		//Wait for Delay, copy Data and then next step
		IF NOT fbMBRead_FC3.bBusy AND NOT fbMBRead_FC3.bError AND timDelay.Q THEN
			// convert received data
			FB_ConvertData(	arrBuffer_FC3			:=	arrBuffer_FC3,
											int_Poll_Counter		:=	int_Poll_Counter,
											lrPowerTotal			=>	fbMeter[int_Poll_Counter].lrPowerTotal,	
											lrReactivePowerTotal	=> 	fbMeter[int_Poll_Counter].lrReactivePowerTotal,
											eOperatingStateInverter	=>	st_Huawei_SmartLogger[int_Poll_Counter].eOperatingStateInverter);
	
			//Next Step
			fbMBRead_FC3.bExecute := FALSE;
			timDelay.IN := FALSE;
			iStateModbus := iStateModbus+1;
			IF arrBuffer_FC3[9]<>0 THEN
				st_Huawei_SmartLogger[int_Poll_Counter].bError := FALSE; 
				st_Huawei_SmartLogger[int_Poll_Counter].eErrorState := E_Huawei_SmartLogger_Error.eNoError;
			ELSE
				st_Huawei_SmartLogger[int_Poll_Counter].bError := FALSE; 
				st_Huawei_SmartLogger[int_Poll_Counter].eErrorState := E_Huawei_SmartLogger_Error.eNoError;
			END_IF
		END_IF
			
		//Error from Inverter 
		IF NOT fbMBRead_FC3.bBusy AND NOT fbMBRead_FC3.bError AND timDelay.Q AND arrBuffer_FC3[9] >= 16#0300 AND arrBuffer_FC3[9] <= 16#0308 THEN
			iStateModbus := 300;
			st_Huawei_SmartLogger[int_Poll_Counter].eErrorState := E_Huawei_SmartLogger_Error.eHuawei_SmartLoggerError;
		END_IF
	
		//Error or Timeout
		IF FPError_FC_3.Q OR timTimeout.Q THEN
			iStateModbus := 300;
			st_Huawei_SmartLogger[int_Poll_Counter].eOperatingStateInverter := E_Huawei_SmartLogger_OperatingState.Unknown;
			st_Huawei_SmartLogger[int_Poll_Counter].eErrorState	:=	E_Huawei_SmartLogger_Error.eModbusTCPError;
		END_IF
		
	2://Wait and go to step 1 or step 3
		iStateModbus_CP := iStateModbus;
		IF sint_ID_Iverter[int_Poll_Counter+1] = 0 OR int_Poll_Counter=int_maxPolls THEN		// if ID is not in use, go to state 100
			iStateModbus := 100;
		ELSE
			iStateModbus := 3;
			int_Poll_Counter:=int_Poll_Counter+1;			//Poll int_Poll_Counter : Inverter int_Poll_Counter 	
		END_IF

	3://Read out next inverter
		st_Huawei_SmartLogger[int_Poll_Counter].bFunctionIsActive := TRUE;
		iStateModbus_CP := iStateModbus;
		fbMBRead_FC3.nQuantity := 25;
		fbMBRead_FC3.nMBAddr := (51000+(25*(SINT_TO_WORD(sint_ID_Iverter[int_Poll_Counter]) - 1)));
		fbMBRead_FC3.bExecute := TRUE;
			
		IF fbMBRead_FC3.bBusy THEN 
			timDelay.IN := TRUE; 
		END_IF
		
		//Wait for Delay, copy Data and then next step
		IF NOT fbMBRead_FC3.bBusy AND NOT fbMBRead_FC3.bError AND timDelay.Q THEN
			// convert received data
			FB_ConvertData(	arrBuffer_FC3			:=	arrBuffer_FC3,
											int_Poll_Counter		:=	int_Poll_Counter,
											lrPowerTotal			=>	fbMeter[int_Poll_Counter].lrPowerTotal,	
											lrReactivePowerTotal	=> 	fbMeter[int_Poll_Counter].lrReactivePowerTotal,
											eOperatingStateInverter	=>	st_Huawei_SmartLogger[int_Poll_Counter].eOperatingStateInverter);
	
			//Next Step
			fbMBRead_FC3.bExecute := FALSE;
			timDelay.IN := FALSE;
			iStateModbus := iStateModbus+1;
			IF arrBuffer_FC3[9]<>0 THEN
				st_Huawei_SmartLogger[int_Poll_Counter].bError := FALSE; 
				st_Huawei_SmartLogger[int_Poll_Counter].eErrorState := E_Huawei_SmartLogger_Error.eNoError;
			ELSE
				st_Huawei_SmartLogger[int_Poll_Counter].bError := FALSE; 
				st_Huawei_SmartLogger[int_Poll_Counter].eErrorState := E_Huawei_SmartLogger_Error.eNoError;
			END_IF
		END_IF
			
		//Error from Inverter 
		IF NOT fbMBRead_FC3.bBusy AND NOT fbMBRead_FC3.bError AND timDelay.Q AND arrBuffer_FC3[9] >= 16#0300 AND arrBuffer_FC3[9] <= 16#0308 THEN
			iStateModbus := 300;
			st_Huawei_SmartLogger[int_Poll_Counter].eErrorState := E_Huawei_SmartLogger_Error.eHuawei_SmartLoggerError;
		END_IF
	
		//Error or Timeout
		IF FPError_FC_3.Q OR timTimeout.Q THEN
			iStateModbus := 300;
			st_Huawei_SmartLogger[int_Poll_Counter].eOperatingStateInverter := E_Huawei_SmartLogger_OperatingState.Unknown;
			st_Huawei_SmartLogger[int_Poll_Counter].eErrorState	:=	E_Huawei_SmartLogger_Error.eModbusTCPError;
		END_IF
		
	4://Wait and go to step +1 or step 100
		iStateModbus_CP := iStateModbus;
		IF sint_ID_Iverter[int_Poll_Counter+1] = 0 OR int_Poll_Counter=int_maxPolls THEN		// if ID is not in use, go to state 100
			iStateModbus := 100;
		ELSE
			iStateModbus := iStateModbus+1;
			int_Poll_Counter:=int_Poll_Counter+1;			//Poll int_Poll_Counter : Inverter int_Poll_Counter 	
		END_IF
	
	5://Read out next inverter
		st_Huawei_SmartLogger[int_Poll_Counter].bFunctionIsActive := TRUE;
		iStateModbus_CP := iStateModbus;
		fbMBRead_FC3.nQuantity := 25;
		fbMBRead_FC3.nMBAddr := (51000+(25*(SINT_TO_WORD(sint_ID_Iverter[int_Poll_Counter]) - 1)));
		fbMBRead_FC3.bExecute := TRUE;
			
		IF fbMBRead_FC3.bBusy THEN 
			timDelay.IN := TRUE; 
		END_IF
		
		//Wait for Delay, copy Data and then next step
		IF NOT fbMBRead_FC3.bBusy AND NOT fbMBRead_FC3.bError AND timDelay.Q THEN
			// convert received data
			FB_ConvertData(	arrBuffer_FC3			:=	arrBuffer_FC3,
											int_Poll_Counter		:=	int_Poll_Counter,
											lrPowerTotal			=>	fbMeter[int_Poll_Counter].lrPowerTotal,	
											lrReactivePowerTotal	=> 	fbMeter[int_Poll_Counter].lrReactivePowerTotal,
											eOperatingStateInverter	=>	st_Huawei_SmartLogger[int_Poll_Counter].eOperatingStateInverter);
	
			//Next Step
			fbMBRead_FC3.bExecute := FALSE;
			timDelay.IN := FALSE;
			iStateModbus := iStateModbus+1;
			IF arrBuffer_FC3[9]<>0 THEN
				st_Huawei_SmartLogger[int_Poll_Counter].bError := FALSE; 
				st_Huawei_SmartLogger[int_Poll_Counter].eErrorState := E_Huawei_SmartLogger_Error.eNoError;
			ELSE
				st_Huawei_SmartLogger[int_Poll_Counter].bError := FALSE; 
				st_Huawei_SmartLogger[int_Poll_Counter].eErrorState := E_Huawei_SmartLogger_Error.eNoError;
			END_IF
		END_IF
			
		//Error from Inverter 
		IF NOT fbMBRead_FC3.bBusy AND NOT fbMBRead_FC3.bError AND timDelay.Q AND arrBuffer_FC3[9] >= 16#0300 AND arrBuffer_FC3[9] <= 16#0308 THEN
			iStateModbus := 300;
			st_Huawei_SmartLogger[int_Poll_Counter].eErrorState := E_Huawei_SmartLogger_Error.eHuawei_SmartLoggerError;
		END_IF
	
		//Error or Timeout
		IF FPError_FC_3.Q OR timTimeout.Q THEN
			iStateModbus := 300;
			st_Huawei_SmartLogger[int_Poll_Counter].eOperatingStateInverter := E_Huawei_SmartLogger_OperatingState.Unknown;
			st_Huawei_SmartLogger[int_Poll_Counter].eErrorState	:=	E_Huawei_SmartLogger_Error.eModbusTCPError;
		END_IF
		
	6://Wait and go to step +1 or step 100
		iStateModbus_CP := iStateModbus;
		IF sint_ID_Iverter[int_Poll_Counter+1] = 0 OR int_Poll_Counter=int_maxPolls THEN		// if ID is not in use, go to state 100
			iStateModbus := 100;
		ELSE
			iStateModbus := iStateModbus+1;
			int_Poll_Counter:=int_Poll_Counter+1;			//Poll int_Poll_Counter : Inverter int_Poll_Counter 	
		END_IF
		
	7://Read out next inverter
		st_Huawei_SmartLogger[int_Poll_Counter].bFunctionIsActive := TRUE;
		iStateModbus_CP := iStateModbus;
		fbMBRead_FC3.nQuantity := 25;
		fbMBRead_FC3.nMBAddr := (51000+(25*(SINT_TO_WORD(sint_ID_Iverter[int_Poll_Counter]) - 1)));
		fbMBRead_FC3.bExecute := TRUE;
			
		IF fbMBRead_FC3.bBusy THEN 
			timDelay.IN := TRUE; 
		END_IF
		
		//Wait for Delay, copy Data and then next step
		IF NOT fbMBRead_FC3.bBusy AND NOT fbMBRead_FC3.bError AND timDelay.Q THEN
			// convert received data
			FB_ConvertData(	arrBuffer_FC3			:=	arrBuffer_FC3,
											int_Poll_Counter		:=	int_Poll_Counter,
											lrPowerTotal			=>	fbMeter[int_Poll_Counter].lrPowerTotal,	
											lrReactivePowerTotal	=> 	fbMeter[int_Poll_Counter].lrReactivePowerTotal,
											eOperatingStateInverter	=>	st_Huawei_SmartLogger[int_Poll_Counter].eOperatingStateInverter);
	
			//Next Step
			fbMBRead_FC3.bExecute := FALSE;
			timDelay.IN := FALSE;
			iStateModbus := iStateModbus+1;
			IF arrBuffer_FC3[9]<>0 THEN
				st_Huawei_SmartLogger[int_Poll_Counter].bError := FALSE; 
				st_Huawei_SmartLogger[int_Poll_Counter].eErrorState := E_Huawei_SmartLogger_Error.eNoError;
			ELSE
				st_Huawei_SmartLogger[int_Poll_Counter].bError := FALSE; 
				st_Huawei_SmartLogger[int_Poll_Counter].eErrorState := E_Huawei_SmartLogger_Error.eNoError;
			END_IF
		END_IF
			
		//Error from Inverter 
		IF NOT fbMBRead_FC3.bBusy AND NOT fbMBRead_FC3.bError AND timDelay.Q AND arrBuffer_FC3[9] >= 16#0300 AND arrBuffer_FC3[9] <= 16#0308 THEN
			iStateModbus := 300;
			st_Huawei_SmartLogger[int_Poll_Counter].eErrorState := E_Huawei_SmartLogger_Error.eHuawei_SmartLoggerError;
		END_IF
	
		//Error or Timeout
		IF FPError_FC_3.Q OR timTimeout.Q THEN
			iStateModbus := 300;
			st_Huawei_SmartLogger[int_Poll_Counter].eOperatingStateInverter := E_Huawei_SmartLogger_OperatingState.Unknown;
			st_Huawei_SmartLogger[int_Poll_Counter].eErrorState	:=	E_Huawei_SmartLogger_Error.eModbusTCPError;
		END_IF

	8://Wait and go to step +1 or step 100
		iStateModbus_CP := iStateModbus;
		IF sint_ID_Iverter[int_Poll_Counter+1] = 0 OR int_Poll_Counter=int_maxPolls THEN		// if ID is not in use, go to state 100
			iStateModbus := 100;
		ELSE
			iStateModbus := iStateModbus+1;
			int_Poll_Counter:=int_Poll_Counter+1;			//Poll int_Poll_Counter : Inverter int_Poll_Counter 	
		END_IF
		
	9://Read out next inverter
		st_Huawei_SmartLogger[int_Poll_Counter].bFunctionIsActive := TRUE;
		iStateModbus_CP := iStateModbus;
		fbMBRead_FC3.nQuantity := 25;
		fbMBRead_FC3.nMBAddr := (51000+(25*(SINT_TO_WORD(sint_ID_Iverter[int_Poll_Counter]) - 1)));
		fbMBRead_FC3.bExecute := TRUE;
			
		IF fbMBRead_FC3.bBusy THEN 
			timDelay.IN := TRUE; 
		END_IF
		
		//Wait for Delay, copy Data and then next step
		IF NOT fbMBRead_FC3.bBusy AND NOT fbMBRead_FC3.bError AND timDelay.Q THEN
			// convert received data
			FB_ConvertData(	arrBuffer_FC3			:=	arrBuffer_FC3,
											int_Poll_Counter		:=	int_Poll_Counter,
											lrPowerTotal			=>	fbMeter[int_Poll_Counter].lrPowerTotal,	
											lrReactivePowerTotal	=> 	fbMeter[int_Poll_Counter].lrReactivePowerTotal,
											eOperatingStateInverter	=>	st_Huawei_SmartLogger[int_Poll_Counter].eOperatingStateInverter);
	
			//Next Step
			fbMBRead_FC3.bExecute := FALSE;
			timDelay.IN := FALSE;
			iStateModbus := iStateModbus+1;
			IF arrBuffer_FC3[9]<>0 THEN
				st_Huawei_SmartLogger[int_Poll_Counter].bError := FALSE; 
				st_Huawei_SmartLogger[int_Poll_Counter].eErrorState := E_Huawei_SmartLogger_Error.eNoError;
			ELSE
				st_Huawei_SmartLogger[int_Poll_Counter].bError := FALSE; 
				st_Huawei_SmartLogger[int_Poll_Counter].eErrorState := E_Huawei_SmartLogger_Error.eNoError;
			END_IF
		END_IF
			
		//Error from Inverter 
		IF NOT fbMBRead_FC3.bBusy AND NOT fbMBRead_FC3.bError AND timDelay.Q AND arrBuffer_FC3[9] >= 16#0300 AND arrBuffer_FC3[9] <= 16#0308 THEN
			iStateModbus := 300;
			st_Huawei_SmartLogger[int_Poll_Counter].eErrorState := E_Huawei_SmartLogger_Error.eHuawei_SmartLoggerError;
		END_IF
	
		//Error or Timeout
		IF FPError_FC_3.Q OR timTimeout.Q THEN
			iStateModbus := 300;
			st_Huawei_SmartLogger[int_Poll_Counter].eOperatingStateInverter := E_Huawei_SmartLogger_OperatingState.Unknown;
			st_Huawei_SmartLogger[int_Poll_Counter].eErrorState	:=	E_Huawei_SmartLogger_Error.eModbusTCPError;
		END_IF
		
	10://Wait and go to step +1 or step 100
		iStateModbus_CP := iStateModbus;
		IF sint_ID_Iverter[int_Poll_Counter+1] = 0 OR int_Poll_Counter=int_maxPolls THEN		// if ID is not in use, go to state 100
			iStateModbus := 100;
		ELSE
			iStateModbus := iStateModbus+1;
			int_Poll_Counter:=int_Poll_Counter+1;			//Poll int_Poll_Counter : Inverter int_Poll_Counter 	
		END_IF
		
	11://Read out next inverter
		st_Huawei_SmartLogger[int_Poll_Counter].bFunctionIsActive := TRUE;
		iStateModbus_CP := iStateModbus;
		fbMBRead_FC3.nQuantity := 25;
		fbMBRead_FC3.nMBAddr := (51000+(25*(SINT_TO_WORD(sint_ID_Iverter[int_Poll_Counter]) - 1)));
		fbMBRead_FC3.bExecute := TRUE;
			
		IF fbMBRead_FC3.bBusy THEN 
			timDelay.IN := TRUE; 
		END_IF
		
		//Wait for Delay, copy Data and then next step
		IF NOT fbMBRead_FC3.bBusy AND NOT fbMBRead_FC3.bError AND timDelay.Q THEN
			// convert received data
			FB_ConvertData(	arrBuffer_FC3			:=	arrBuffer_FC3,
											int_Poll_Counter		:=	int_Poll_Counter,
											lrPowerTotal			=>	fbMeter[int_Poll_Counter].lrPowerTotal,	
											lrReactivePowerTotal	=> 	fbMeter[int_Poll_Counter].lrReactivePowerTotal,
											eOperatingStateInverter	=>	st_Huawei_SmartLogger[int_Poll_Counter].eOperatingStateInverter);
	
			//Next Step
			fbMBRead_FC3.bExecute := FALSE;
			timDelay.IN := FALSE;
			iStateModbus := iStateModbus+1;
			IF arrBuffer_FC3[9]<>0 THEN
				st_Huawei_SmartLogger[int_Poll_Counter].bError := FALSE; 
				st_Huawei_SmartLogger[int_Poll_Counter].eErrorState := E_Huawei_SmartLogger_Error.eNoError;
			ELSE
				st_Huawei_SmartLogger[int_Poll_Counter].bError := FALSE; 
				st_Huawei_SmartLogger[int_Poll_Counter].eErrorState := E_Huawei_SmartLogger_Error.eNoError;
			END_IF
		END_IF
			
		//Error from Inverter 
		IF NOT fbMBRead_FC3.bBusy AND NOT fbMBRead_FC3.bError AND timDelay.Q AND arrBuffer_FC3[9] >= 16#0300 AND arrBuffer_FC3[9] <= 16#0308 THEN
			iStateModbus := 300;
			st_Huawei_SmartLogger[int_Poll_Counter].eErrorState := E_Huawei_SmartLogger_Error.eHuawei_SmartLoggerError;
		END_IF
	
		//Error or Timeout
		IF FPError_FC_3.Q OR timTimeout.Q THEN
			iStateModbus := 300;
			st_Huawei_SmartLogger[int_Poll_Counter].eOperatingStateInverter := E_Huawei_SmartLogger_OperatingState.Unknown;
			st_Huawei_SmartLogger[int_Poll_Counter].eErrorState	:=	E_Huawei_SmartLogger_Error.eModbusTCPError;
		END_IF
		
	12://Wait and go to step +1 or step 100
		iStateModbus_CP := iStateModbus;
		IF sint_ID_Iverter[int_Poll_Counter+1] = 0 OR int_Poll_Counter=int_maxPolls THEN		// if ID is not in use, go to state 100
			iStateModbus := 100;
		ELSE
			iStateModbus := iStateModbus+1;
			int_Poll_Counter:=int_Poll_Counter+1;			//Poll int_Poll_Counter : Inverter int_Poll_Counter 	
		END_IF
		
	13://Read out next inverter
		st_Huawei_SmartLogger[int_Poll_Counter].bFunctionIsActive := TRUE;
		iStateModbus_CP := iStateModbus;
		fbMBRead_FC3.nQuantity := 25;
		fbMBRead_FC3.nMBAddr := (51000+(25*(SINT_TO_WORD(sint_ID_Iverter[int_Poll_Counter]) - 1)));
		fbMBRead_FC3.bExecute := TRUE;
			
		IF fbMBRead_FC3.bBusy THEN 
			timDelay.IN := TRUE; 
		END_IF
		
		//Wait for Delay, copy Data and then next step
		IF NOT fbMBRead_FC3.bBusy AND NOT fbMBRead_FC3.bError AND timDelay.Q THEN
			// convert received data
			FB_ConvertData(	arrBuffer_FC3			:=	arrBuffer_FC3,
											int_Poll_Counter		:=	int_Poll_Counter,
											lrPowerTotal			=>	fbMeter[int_Poll_Counter].lrPowerTotal,	
											lrReactivePowerTotal	=> 	fbMeter[int_Poll_Counter].lrReactivePowerTotal,
											eOperatingStateInverter	=>	st_Huawei_SmartLogger[int_Poll_Counter].eOperatingStateInverter);
	
			//Next Step
			fbMBRead_FC3.bExecute := FALSE;
			timDelay.IN := FALSE;
			iStateModbus := iStateModbus+1;
			IF arrBuffer_FC3[9]<>0 THEN
				st_Huawei_SmartLogger[int_Poll_Counter].bError := FALSE; 
				st_Huawei_SmartLogger[int_Poll_Counter].eErrorState := E_Huawei_SmartLogger_Error.eNoError;
			ELSE
				st_Huawei_SmartLogger[int_Poll_Counter].bError := FALSE; 
				st_Huawei_SmartLogger[int_Poll_Counter].eErrorState := E_Huawei_SmartLogger_Error.eNoError;
			END_IF
		END_IF
			
		//Error from Inverter 1
		IF NOT fbMBRead_FC3.bBusy AND NOT fbMBRead_FC3.bError AND timDelay.Q AND arrBuffer_FC3[9] >= 16#0300 AND arrBuffer_FC3[9] <= 16#0308 THEN
			iStateModbus := 300;
			st_Huawei_SmartLogger[int_Poll_Counter].eErrorState := E_Huawei_SmartLogger_Error.eHuawei_SmartLoggerError;
		END_IF
	
		//Error or Timeout
		IF FPError_FC_3.Q OR timTimeout.Q THEN
			iStateModbus := 300;
			st_Huawei_SmartLogger[int_Poll_Counter].eOperatingStateInverter := E_Huawei_SmartLogger_OperatingState.Unknown;
			st_Huawei_SmartLogger[int_Poll_Counter].eErrorState	:=	E_Huawei_SmartLogger_Error.eModbusTCPError;
		END_IF
		
	14://Wait and go to step +1 or step 100
		iStateModbus_CP := iStateModbus;
		IF sint_ID_Iverter[int_Poll_Counter+1] = 0 OR int_Poll_Counter=int_maxPolls THEN		// if ID is not in use, go to state 100
			iStateModbus := 100;
		ELSE
			iStateModbus := iStateModbus+1;
			int_Poll_Counter:=int_Poll_Counter+1;			//Poll int_Poll_Counter : Inverter int_Poll_Counter 	
		END_IF
		
	15://Read out next inverter
		st_Huawei_SmartLogger[int_Poll_Counter].bFunctionIsActive := TRUE;
		iStateModbus_CP := iStateModbus;
		fbMBRead_FC3.nQuantity := 25;
		fbMBRead_FC3.nMBAddr := (51000+(25*(SINT_TO_WORD(sint_ID_Iverter[int_Poll_Counter]) - 1)));
		fbMBRead_FC3.bExecute := TRUE;
			
		IF fbMBRead_FC3.bBusy THEN 
			timDelay.IN := TRUE; 
		END_IF
		
		//Wait for Delay, copy Data and then next step
		IF NOT fbMBRead_FC3.bBusy AND NOT fbMBRead_FC3.bError AND timDelay.Q THEN
			// convert received data
			FB_ConvertData(	arrBuffer_FC3			:=	arrBuffer_FC3,
											int_Poll_Counter		:=	int_Poll_Counter,
											lrPowerTotal			=>	fbMeter[int_Poll_Counter].lrPowerTotal,	
											lrReactivePowerTotal	=> 	fbMeter[int_Poll_Counter].lrReactivePowerTotal,
											eOperatingStateInverter	=>	st_Huawei_SmartLogger[int_Poll_Counter].eOperatingStateInverter);
	
			//Next Step
			fbMBRead_FC3.bExecute := FALSE;
			timDelay.IN := FALSE;
			iStateModbus := iStateModbus+1;
			IF arrBuffer_FC3[9]<>0 THEN
				st_Huawei_SmartLogger[int_Poll_Counter].bError := FALSE; 
				st_Huawei_SmartLogger[int_Poll_Counter].eErrorState := E_Huawei_SmartLogger_Error.eNoError;
			ELSE
				st_Huawei_SmartLogger[int_Poll_Counter].bError := FALSE; 
				st_Huawei_SmartLogger[int_Poll_Counter].eErrorState := E_Huawei_SmartLogger_Error.eNoError;
			END_IF
		END_IF
			
		//Error from Inverter 
		IF NOT fbMBRead_FC3.bBusy AND NOT fbMBRead_FC3.bError AND timDelay.Q AND arrBuffer_FC3[9] >= 16#0300 AND arrBuffer_FC3[9] <= 16#0308 THEN
			iStateModbus := 300;
			st_Huawei_SmartLogger[int_Poll_Counter].eErrorState := E_Huawei_SmartLogger_Error.eHuawei_SmartLoggerError;
		END_IF
	
		//Error or Timeout
		IF FPError_FC_3.Q OR timTimeout.Q THEN
			iStateModbus := 300;
			st_Huawei_SmartLogger[int_Poll_Counter].eOperatingStateInverter := E_Huawei_SmartLogger_OperatingState.Unknown;
			st_Huawei_SmartLogger[int_Poll_Counter].eErrorState	:=	E_Huawei_SmartLogger_Error.eModbusTCPError;
		END_IF
		
	16://Wait and go to step +1 or step 100
		iStateModbus_CP := iStateModbus;
		IF sint_ID_Iverter[int_Poll_Counter+1] = 0 OR int_Poll_Counter=int_maxPolls THEN		// if ID is not in use, go to state 100
			iStateModbus := 100;
		ELSE
			iStateModbus := iStateModbus+1;
			int_Poll_Counter:=int_Poll_Counter+1;			//Poll int_Poll_Counter : Inverter int_Poll_Counter 	
		END_IF

	17://Read out next inverter
		st_Huawei_SmartLogger[int_Poll_Counter].bFunctionIsActive := TRUE;
		iStateModbus_CP := iStateModbus;
		fbMBRead_FC3.nQuantity := 25;
		fbMBRead_FC3.nMBAddr := (51000+(25*(SINT_TO_WORD(sint_ID_Iverter[int_Poll_Counter]) - 1)));
		fbMBRead_FC3.bExecute := TRUE;
			
		IF fbMBRead_FC3.bBusy THEN 
			timDelay.IN := TRUE; 
		END_IF
		
		//Wait for Delay, copy Data and then next step
		IF NOT fbMBRead_FC3.bBusy AND NOT fbMBRead_FC3.bError AND timDelay.Q THEN
			// convert received data
			FB_ConvertData(	arrBuffer_FC3			:=	arrBuffer_FC3,
											int_Poll_Counter		:=	int_Poll_Counter,
											lrPowerTotal			=>	fbMeter[int_Poll_Counter].lrPowerTotal,	
											lrReactivePowerTotal	=> 	fbMeter[int_Poll_Counter].lrReactivePowerTotal,
											eOperatingStateInverter	=>	st_Huawei_SmartLogger[int_Poll_Counter].eOperatingStateInverter);
	
			//Next Step
			fbMBRead_FC3.bExecute := FALSE;
			timDelay.IN := FALSE;
			iStateModbus := iStateModbus+1;
			IF arrBuffer_FC3[9]<>0 THEN
				st_Huawei_SmartLogger[int_Poll_Counter].bError := FALSE; 
				st_Huawei_SmartLogger[int_Poll_Counter].eErrorState := E_Huawei_SmartLogger_Error.eNoError;
			ELSE
				st_Huawei_SmartLogger[int_Poll_Counter].bError := FALSE; 
				st_Huawei_SmartLogger[int_Poll_Counter].eErrorState := E_Huawei_SmartLogger_Error.eNoError;
			END_IF
		END_IF
			
		//Error from Inverter 
		IF NOT fbMBRead_FC3.bBusy AND NOT fbMBRead_FC3.bError AND timDelay.Q AND arrBuffer_FC3[9] >= 16#0300 AND arrBuffer_FC3[9] <= 16#0308 THEN
			iStateModbus := 300;
			st_Huawei_SmartLogger[int_Poll_Counter].eErrorState := E_Huawei_SmartLogger_Error.eHuawei_SmartLoggerError;
		END_IF
	
		//Error or Timeout
		IF FPError_FC_3.Q OR timTimeout.Q THEN
			iStateModbus := 300;
			st_Huawei_SmartLogger[int_Poll_Counter].eOperatingStateInverter := E_Huawei_SmartLogger_OperatingState.Unknown;
			st_Huawei_SmartLogger[int_Poll_Counter].eErrorState	:=	E_Huawei_SmartLogger_Error.eModbusTCPError;
		END_IF
		
	18://Wait and go to step +1 or step 100
		iStateModbus_CP := iStateModbus;
		IF sint_ID_Iverter[int_Poll_Counter+1] = 0 OR int_Poll_Counter=int_maxPolls THEN		// if ID is not in use, go to state 100
			iStateModbus := 100;
		ELSE
			iStateModbus := iStateModbus+1;
			int_Poll_Counter:=int_Poll_Counter+1;			//Poll int_Poll_Counter : Inverter int_Poll_Counter 	
		END_IF
		
	19://Read out next inverter
		st_Huawei_SmartLogger[int_Poll_Counter].bFunctionIsActive := TRUE;
		iStateModbus_CP := iStateModbus;
		fbMBRead_FC3.nQuantity := 25;
		fbMBRead_FC3.nMBAddr := (51000+(25*(SINT_TO_WORD(sint_ID_Iverter[int_Poll_Counter]) - 1)));
		fbMBRead_FC3.bExecute := TRUE;
			
		IF fbMBRead_FC3.bBusy THEN 
			timDelay.IN := TRUE; 
		END_IF
		
		//Wait for Delay, copy Data and then next step
		IF NOT fbMBRead_FC3.bBusy AND NOT fbMBRead_FC3.bError AND timDelay.Q THEN
			// convert received data
			FB_ConvertData(	arrBuffer_FC3			:=	arrBuffer_FC3,
											int_Poll_Counter		:=	int_Poll_Counter,
											lrPowerTotal			=>	fbMeter[int_Poll_Counter].lrPowerTotal,	
											lrReactivePowerTotal	=> 	fbMeter[int_Poll_Counter].lrReactivePowerTotal,
											eOperatingStateInverter	=>	st_Huawei_SmartLogger[int_Poll_Counter].eOperatingStateInverter);
	
			//Next Step
			fbMBRead_FC3.bExecute := FALSE;
			timDelay.IN := FALSE;
			iStateModbus := iStateModbus+1;
			IF arrBuffer_FC3[9]<>0 THEN
				st_Huawei_SmartLogger[int_Poll_Counter].bError := FALSE; 
				st_Huawei_SmartLogger[int_Poll_Counter].eErrorState := E_Huawei_SmartLogger_Error.eNoError;
			ELSE
				st_Huawei_SmartLogger[int_Poll_Counter].bError := FALSE; 
				st_Huawei_SmartLogger[int_Poll_Counter].eErrorState := E_Huawei_SmartLogger_Error.eNoError;
			END_IF
		END_IF
			
		//Error or Timeout
		IF FPError_FC_3.Q OR timTimeout.Q THEN
			iStateModbus := 300;
			st_Huawei_SmartLogger[int_Poll_Counter].eOperatingStateInverter := E_Huawei_SmartLogger_OperatingState.Unknown;
			st_Huawei_SmartLogger[int_Poll_Counter].eErrorState	:=	E_Huawei_SmartLogger_Error.eModbusTCPError;
		END_IF
	
		//Error or Timeout
		IF FPError_FC_3.Q OR timTimeout.Q THEN
			iStateModbus := 300;
			st_Huawei_SmartLogger[int_Poll_Counter].eOperatingStateInverter := E_Huawei_SmartLogger_Error.eModbusTCPError;
		END_IF

	20://Wait and go to step +1 or step 100
		iStateModbus_CP := iStateModbus;
		IF sint_ID_Iverter[int_Poll_Counter+1] = 0 OR int_Poll_Counter=int_maxPolls THEN		// if ID is not in use, go to state 100
			iStateModbus := 100;
		ELSE
			iStateModbus := iStateModbus+1;
			int_Poll_Counter:=int_Poll_Counter+1;			//Poll int_Poll_Counter : Inverter int_Poll_Counter 	
		END_IF

	21://Read out next inverter
		st_Huawei_SmartLogger[int_Poll_Counter].bFunctionIsActive := TRUE;
		iStateModbus_CP := iStateModbus;
		fbMBRead_FC3.nQuantity := 25;
		fbMBRead_FC3.nMBAddr := (51000+(25*(SINT_TO_WORD(sint_ID_Iverter[int_Poll_Counter]) - 1)));
		fbMBRead_FC3.bExecute := TRUE;
			
		IF fbMBRead_FC3.bBusy THEN 
			timDelay.IN := TRUE; 
		END_IF
		
		//Wait for Delay, copy Data and then next step
		IF NOT fbMBRead_FC3.bBusy AND NOT fbMBRead_FC3.bError AND timDelay.Q THEN
			// convert received data
			FB_ConvertData(	arrBuffer_FC3			:=	arrBuffer_FC3,
											int_Poll_Counter		:=	int_Poll_Counter,
											lrPowerTotal			=>	fbMeter[int_Poll_Counter].lrPowerTotal,	
											lrReactivePowerTotal	=> 	fbMeter[int_Poll_Counter].lrReactivePowerTotal,
											eOperatingStateInverter	=>	st_Huawei_SmartLogger[int_Poll_Counter].eOperatingStateInverter);
	
			//Next Step
			fbMBRead_FC3.bExecute := FALSE;
			timDelay.IN := FALSE;
			iStateModbus := iStateModbus+1;
			IF arrBuffer_FC3[9]<>0 THEN
				st_Huawei_SmartLogger[int_Poll_Counter].bError := FALSE; 
				st_Huawei_SmartLogger[int_Poll_Counter].eErrorState := E_Huawei_SmartLogger_Error.eNoError;
			ELSE
				st_Huawei_SmartLogger[int_Poll_Counter].bError := FALSE; 
				st_Huawei_SmartLogger[int_Poll_Counter].eErrorState := E_Huawei_SmartLogger_Error.eNoError;
			END_IF
		END_IF
			
		//Error from Inverter 
		IF NOT fbMBRead_FC3.bBusy AND NOT fbMBRead_FC3.bError AND timDelay.Q AND arrBuffer_FC3[9] >= 16#0300 AND arrBuffer_FC3[9] <= 16#0308 THEN
			iStateModbus := 300;
			st_Huawei_SmartLogger[int_Poll_Counter].eErrorState := E_Huawei_SmartLogger_Error.eHuawei_SmartLoggerError;
		END_IF
	
		//Error or Timeout
		IF FPError_FC_3.Q OR timTimeout.Q THEN
			iStateModbus := 300;
			st_Huawei_SmartLogger[int_Poll_Counter].eOperatingStateInverter := E_Huawei_SmartLogger_OperatingState.Unknown;
			st_Huawei_SmartLogger[int_Poll_Counter].eErrorState	:=	E_Huawei_SmartLogger_Error.eModbusTCPError;
		END_IF
		
	22://Wait and go to step +1 or step 100
		iStateModbus_CP := iStateModbus;
		IF sint_ID_Iverter[int_Poll_Counter+1] = 0 OR int_Poll_Counter=int_maxPolls THEN		// if ID is not in use, go to state 100
			iStateModbus := 100;
		ELSE
			iStateModbus := iStateModbus+1;
			int_Poll_Counter:=int_Poll_Counter+1;			//Poll int_Poll_Counter : Inverter int_Poll_Counter 	
		END_IF

	23://Read out next inverter
		st_Huawei_SmartLogger[int_Poll_Counter].bFunctionIsActive := TRUE;
		iStateModbus_CP := iStateModbus;
		fbMBRead_FC3.nQuantity := 25;
		fbMBRead_FC3.nMBAddr := (51000+(25*(SINT_TO_WORD(sint_ID_Iverter[int_Poll_Counter]) - 1)));
		fbMBRead_FC3.bExecute := TRUE;
			
		IF fbMBRead_FC3.bBusy THEN 
			timDelay.IN := TRUE; 
		END_IF
		
		//Wait for Delay, copy Data and then next step
		IF NOT fbMBRead_FC3.bBusy AND NOT fbMBRead_FC3.bError AND timDelay.Q THEN
			// convert received data
			FB_ConvertData(	arrBuffer_FC3			:=	arrBuffer_FC3,
											int_Poll_Counter		:=	int_Poll_Counter,
											lrPowerTotal			=>	fbMeter[int_Poll_Counter].lrPowerTotal,	
											lrReactivePowerTotal	=> 	fbMeter[int_Poll_Counter].lrReactivePowerTotal,
											eOperatingStateInverter	=>	st_Huawei_SmartLogger[int_Poll_Counter].eOperatingStateInverter);
	
			//Next Step
			fbMBRead_FC3.bExecute := FALSE;
			timDelay.IN := FALSE;
			iStateModbus := iStateModbus+1;
			IF arrBuffer_FC3[9]<>0 THEN
				st_Huawei_SmartLogger[int_Poll_Counter].bError := FALSE; 
				st_Huawei_SmartLogger[int_Poll_Counter].eErrorState := E_Huawei_SmartLogger_Error.eNoError;
			ELSE
				st_Huawei_SmartLogger[int_Poll_Counter].bError := FALSE; 
				st_Huawei_SmartLogger[int_Poll_Counter].eErrorState := E_Huawei_SmartLogger_Error.eNoError;
			END_IF
		END_IF
			
		//Error from Inverter 
		IF NOT fbMBRead_FC3.bBusy AND NOT fbMBRead_FC3.bError AND timDelay.Q AND arrBuffer_FC3[9] >= 16#0300 AND arrBuffer_FC3[9] <= 16#0308 THEN
			iStateModbus := 300;
			st_Huawei_SmartLogger[int_Poll_Counter].eErrorState := E_Huawei_SmartLogger_Error.eHuawei_SmartLoggerError;
		END_IF
	
		//Error or Timeout
		IF FPError_FC_3.Q OR timTimeout.Q THEN
			iStateModbus := 300;
			st_Huawei_SmartLogger[int_Poll_Counter].eOperatingStateInverter := E_Huawei_SmartLogger_OperatingState.Unknown;
			st_Huawei_SmartLogger[int_Poll_Counter].eErrorState	:=	E_Huawei_SmartLogger_Error.eModbusTCPError;
		END_IF
		
	24://Wait and go to step +1 or step 100
		iStateModbus_CP := iStateModbus;
		IF sint_ID_Iverter[int_Poll_Counter+1] = 0 OR int_Poll_Counter=int_maxPolls THEN		// if ID is not in use, go to state 100
			iStateModbus := 100;
		ELSE
			iStateModbus := iStateModbus+1;
			int_Poll_Counter:=int_Poll_Counter+1;			//Poll int_Poll_Counter : Inverter int_Poll_Counter 	
		END_IF




		
		
		
	100://Wait and go to step 1 
		iStateModbus_CP := iStateModbus;
		ton_Wait.In:=TRUE;
		IF ton_Wait.Q THEN
			ton_Wait.In:=FALSE;
			iStateModbus := 1;
		END_IF
			
	300://Error
		iStateModbus_CP := iStateModbus;
		timDelay.IN := FALSE;
		fbMBRead_FC3.bExecute := FALSE;
		st_Huawei_SmartLogger[int_Poll_Counter].bError := TRUE;
		ton_Wait.In:=TRUE;
		IF ton_Wait.Q THEN
			ton_Wait.In:=FALSE;
			iStateModbus := 1;
		END_IF
END_CASE

// wait timer
ton_Wait(PT:=T#2S);

	

(*------------------------------------------------------------------------------------------Modbus TCP Function---------------------------------------------------------------------------------------------*)

fbMBRead_FC3(	sIPAddr:= sIPAdress, 
				nTCPPort:= 502, 
				nUnitID := 0,
				cbLength:= SIZEOF(arrBuffer_FC3), 
				pDestAddr:= ADR(arrBuffer_FC3), 
				tTimeout:= T#10S );

FPError_FC_3(CLK:= fbMBRead_FC3.bError, Q=> );

(*----------------------------------------------------------------------------------------Electric Meter Data----------------------------------------------------------------------------------------------*)

//Error and Warning
FOR x:=1 TO 20 BY 1 DO
	IF timDissableFunctions.Q THEN 
		fbMeter[x].bWarning := TRUE; 
		fbMeter[x].iWarningCode := 0; 
	ELSE 
		fbMeter[x].bWarning := FALSE; 
	END_IF   

	IF st_Huawei_SmartLogger[x].bError OR Lynus_Standards.GVL_Energy.stNumberOfDevices.diNumberOfElectricMeters > Constants_Energy.diMaxNumberOfElectricMeters THEN 
		fbMeter[x].bError := TRUE; 
	ELSE 
		fbMeter[x].bError := FALSE; 
	END_IF  

	IF Lynus_Standards.GVL_Energy.stNumberOfDevices.diNumberOfElectricMeters > Constants_Energy.diMaxNumberOfElectricMeters THEN 
		fbMeter[x].iErrorCode := 1;
	ELSIF st_Huawei_SmartLogger[x].bError THEN 
		fbMeter[x].iErrorCode := 0;
	END_IF  

	//Function block for meter data
	fbMeter[x](
		bEnable:= bEnable AND NOT timDissableFunctions.Q, 
		bError:= , 
		bEnableReadOutFunction:= TRUE, 
		bWriteWithDelay:= TRUE,
		bPowerDataInvers:= TRUE, 
		bReadOutDataDone:= TRUE,
		iTimeReadOutInterval:= , 
		iErrorCode:= , 
		iWarningCode:= , 
		lrTotalCounterEnergy_Consumption:= 0, 
		lrTotalCounterEnergy_Production:= , 
		lrCounterEnergyT1_Consumption:= 0, 
		lrCounterEnergyT2_Consumption:= 0, 
		lrCounterEnergyT1_Production:= , 
		lrCounterEnergyT2_Production:= 0, 
		lrCurrentL1:= , 
		lrVoltageL1N:= , 
		lrVoltageL1L2:= , 
		lrPowerL1:= 0, 
		lrCurrentL2:= , 
		lrVoltageL2N:= , 
		lrVoltageL2L3:= , 
		lrPowerL2:= 0, 
		lrCurrentL3:= , 
		lrVoltageL3N:= , 
		lrVoltageL3L1:= , 
		lrPowerL3:= 0, 
		lrPowerTotal:= , 
		lrFrequency:= , 
		lrReactivePowerTotal:= , 
		lrApparentPowerTotal:= , 
		tTimDelayOutput:= T#5S, 
		stDataEMOutPower=> , 
		stDataEMOutPowerDelay=> stDataEMPower_PV[x], 
		stDataEMOutCounter=> ,
		stDataEMOutCounterDelay=> stDataEMCounter_PV[x], 
		bReadOutMeter=> );

END_FOR
//Read Out Data done for EM Function
IF NOT fbMBRead_FC3.bBusy AND NOT fbMBRead_FC3.bError THEN 
	fbMeter[int_Poll_Counter].bReadOutDataDone := TRUE;
ELSE 
	fbMeter[int_Poll_Counter].bReadOutDataDone := FALSE;
END_IF



(*-----------------------------------------------------------Handle data to Global structure for the Electric Meter system-----------------------------------------------------------------*)

CASE iStateGVLData OF
	
	0://Init Step
		byWaitInStep := 0;
		diCounterForGVL := 1;
	
	1://Wait for 4 Steps before clean al Data on GVL
		byWaitInStep := byWaitInStep + 1;
		IF byWaitInStep >= 4 AND fbNumberDevice.bNumberIsCalculatet THEN 
			iStateGVLData := 2; 
		END_IF
		//To much Devices, back to the Init step
		IF byWaitInStep >= 4 AND NOT fbNumberDevice.bNumberIsCalculatet THEN 
			iStateGVLData := 0; 
		END_IF	
			
	2://Clear all Data in GVL
		Lynus_Standards.GVL_Energy.stDataElectricMeters[diCounterForGVL].bEnabled := FALSE;	
		Lynus_Standards.GVL_Energy.stDataElectricMeters[diCounterForGVL].byErrorWarning := 0;
		Lynus_Standards.GVL_Energy.stDataElectricMeters[diCounterForGVL].lrCounterEnergyT1_Consumption := 0;
		Lynus_Standards.GVL_Energy.stDataElectricMeters[diCounterForGVL].lrCounterEnergyT1_Production := 0;
		Lynus_Standards.GVL_Energy.stDataElectricMeters[diCounterForGVL].lrCounterEnergyT2_Consumption := 0;
		Lynus_Standards.GVL_Energy.stDataElectricMeters[diCounterForGVL].lrCounterEnergyT2_Production := 0;
		Lynus_Standards.GVL_Energy.stDataElectricMeters[diCounterForGVL].lrPower := 0;
		Lynus_Standards.GVL_Energy.stDataElectricMeters[diCounterForGVL].lrPowerConsumption := 0;
		Lynus_Standards.GVL_Energy.stDataElectricMeters[diCounterForGVL].lrPowerConsumption := 0;
		Lynus_Standards.GVL_Energy.stDataElectricMeters[diCounterForGVL].lrPowerProduction := 0;
		Lynus_Standards.GVL_Energy.stDataElectricMeters[diCounterForGVL].lrTotalCounterEnergy_Consumption := 0;
		Lynus_Standards.GVL_Energy.stDataElectricMeters[diCounterForGVL].lrTotalCounterEnergy_Production := 0;
		
		diCounterForGVL := diCounterForGVL + 1;
		diCounterForGVL := LIMIT(0,diCounterForGVL,Constants_Energy.diMaxNumberOfElectricMeters);
		//Back to the init step
		IF diCounterForGVL >= Constants_Energy.diMaxNumberOfElectricMeters THEN 
			iStateGVLData := 0; 
		END_IF
END_CASE 	 

IF diNrOfEM_OUT_PV > 0 AND fbNumberDevice.bNumberIsCalculatet THEN
	Lynus_Standards.GVL_Energy.stDataElectricMeters[diNrOfEM_OUT_PV].bEnabled := fbElMeter.stDataEMOutPower.bEnabled;
	Lynus_Standards.GVL_Energy.stDataElectricMeters[diNrOfEM_OUT_PV].byErrorWarning := fbElMeter.stDataEMOutPower.byErrorWarning;
	Lynus_Standards.GVL_Energy.stDataElectricMeters[diNrOfEM_OUT_PV].lrCounterEnergyT1_Consumption := fbElMeter.stDataEMOutCounter.lrCounterEnergyT1_Consumption;
	Lynus_Standards.GVL_Energy.stDataElectricMeters[diNrOfEM_OUT_PV].lrCounterEnergyT1_Production := fbElMeter.stDataEMOutCounter.lrCounterEnergyT1_Production;
	Lynus_Standards.GVL_Energy.stDataElectricMeters[diNrOfEM_OUT_PV].lrCounterEnergyT2_Consumption := fbElMeter.stDataEMOutCounter.lrCounterEnergyT2_Consumption;
	Lynus_Standards.GVL_Energy.stDataElectricMeters[diNrOfEM_OUT_PV].lrCounterEnergyT2_Production := fbElMeter.stDataEMOutCounter.lrCounterEnergyT2_Production;		
	Lynus_Standards.GVL_Energy.stDataElectricMeters[diNrOfEM_OUT_PV].lrPower := fbElMeter.lrPowerTotal; // fbElMeter.stDataEMOutPower.lrPowerTotal;
	Lynus_Standards.GVL_Energy.stDataElectricMeters[diNrOfEM_OUT_PV].lrPowerConsumption := fbElMeter.stDataEMOutPower.lrPowerConsumption;
	Lynus_Standards.GVL_Energy.stDataElectricMeters[diNrOfEM_OUT_PV].lrPowerProduction := fbElMeter.stDataEMOutPower.lrPowerProduction;
	Lynus_Standards.GVL_Energy.stDataElectricMeters[diNrOfEM_OUT_PV].lrTotalCounterEnergy_Consumption := fbElMeter.stDataEMOutCounter.lrTotalCounterEnergy_Consumption;
	Lynus_Standards.GVL_Energy.stDataElectricMeters[diNrOfEM_OUT_PV].lrTotalCounterEnergy_Production := fbElMeter.stDataEMOutCounter.lrTotalCounterEnergy_Production;
END_IF


// Sum values for Meter
fbElMeter.lrPowerTotal := 0;
FOR byLPForInverter := 1 TO 20 BY 1 DO 
	lrCounterEnergyProduction := lrCounterEnergyProduction + fbMeter[byLPForInverter].stDataEMOutCounterDelay.lrTotalCounterEnergy_Production;
	IF lrCounterEnergyProduction > fbElMeter.lrCounterEnergyT1_Production THEN
		fbElMeter.lrCounterEnergyT1_Production := lrCounterEnergyProduction;
	END_IF
	fbElMeter.lrPowerTotal := fbElMeter.lrPowerTotal + fbMeter[byLPForInverter].stDataEMOutPowerDelay.lrPowerTotal;
END_FOR	
					
fbElMeter.lrTotalCounterEnergy_Production := fbElMeter.lrCounterEnergyT1_Production; 
fbElMeter(bEnable:=TRUE);


lreal1:=fbMeter[1].stDataEMOutPowerDelay.lrPowerTotal;
lreal2:=fbMeter[2].stDataEMOutPowerDelay.lrPowerTotal;
lreal3:=fbMeter[3].stDataEMOutPowerDelay.lrPowerTotal;
lreal4:=fbMeter[4].stDataEMOutPowerDelay.lrPowerTotal;
lreal5:=fbMeter[5].stDataEMOutPowerDelay.lrPowerTotal;
lreal6:=fbMeter[6].stDataEMOutPowerDelay.lrPowerTotal;
lreal7:=fbMeter[7].stDataEMOutPowerDelay.lrPowerTotal;
lreal8:=fbMeter[8].stDataEMOutPowerDelay.lrPowerTotal;
lreal9:=fbMeter[9].stDataEMOutPowerDelay.lrPowerTotal;
lreal10:=fbMeter[10].stDataEMOutPowerDelay.lrPowerTotal;
lreal11:=fbMeter[11].stDataEMOutPowerDelay.lrPowerTotal;
lreal12:=fbMeter[12].stDataEMOutPowerDelay.lrPowerTotal;
lreal13:=fbMeter[13].stDataEMOutPowerDelay.lrPowerTotal;
lreal14:=fbMeter[14].stDataEMOutPowerDelay.lrPowerTotal;
lreal15:=fbMeter[15].stDataEMOutPowerDelay.lrPowerTotal;
lreal16:=fbMeter[16].stDataEMOutPowerDelay.lrPowerTotal;
lreal17:=fbMeter[17].stDataEMOutPowerDelay.lrPowerTotal;
lreal18:=fbMeter[18].stDataEMOutPowerDelay.lrPowerTotal;
lreal19:=fbMeter[19].stDataEMOutPowerDelay.lrPowerTotal;
lreal20:=fbMeter[20].stDataEMOutPowerDelay.lrPowerTotal;

(*----------------------------------------------------------Save persistent data----------------------------------------------------------------*)

// arrPD[1](lrValue:= BOOL_TO_LREAL(bEnable), bEventBasedActive=> );
// arrPD[2](lrValue:= BYTE_TO_LREAL(byAmountOfInverters), bEventBasedActive=> );
PD_String(sText:= sIPAdress, bEventBasedActive=> );

END_FUNCTION_BLOCK

// ---- POUs/prgComEffIO.TcPOU
PROGRAM prgComEffIO
VAR
	fbCom		: FB_MqttCommunicator_V3;
	f_Trig_HB: f_trig;
	stringArray_Last_HB: ARRAY[0..50] OF STRING(30);
	intCount: INT;
	time_Temp: TIME;
	count_u: ctu;
	count_u1: ctu;
	count_u2: ctu;
	
	eErrorMessage_Read				: eErrorMessage;																		//Enum with the Error states
	arrErrorIntern					: ARRAY[0..Constants_Communicator.bySizeOfReceivedValueArrayInJson] OF BOOL;			//Array with Error flag	

	
END_VAR

(*fbCom(
	bConnect:= TRUE,
	strAuthKey := 'EIO08031879806',
	sUserName:= '5ee57453-fd55-4192-b735-1cf18f64f6fd', 
	sUserPassword:= 'f5feda32-4250-448e-ac0f-0ee8f7492652', 
	eSavePositionCertificate:= eSavePositionOnPLC.ePostionHardDisk, 
	bConnected=> , 
	bError=> , 
	hrErrorCode=> , 
	eConnectionState=> , 
	eErrorMessage_Out=> );
*)
fbCom(
	bConnect:= TRUE, 
	strAuthKey:=  'BMS99299754422' , 
	sUserName:= 'a77d1054-48f1-4ad6-a5da-3c6ee387acdf', 
	sUserPassword:= '8404ad90-0db5-41cf-bf43-c0af7cbd8420', 
	eSavePositionCertificate:= eSavePositionOnPLC.ePostionHardDisk,  
	time_HeartBeat_sec 		:= T#15S,
	bConnected=> , 
	bError=> , 
	hrErrorCode=> , 
	eConnectionState=> , 
	eErrorMessage_Out=> );
(*old
	sUserName:= '5ee57453-fd55-4192-b735-1cf18f64f6fd', 
	sUserPassword:= 'f5feda32-4250-448e-ac0f-0ee8f7492652', 
*)
	
f_Trig_HB(CLK :=  fbCom.bHBSending);



prg_SystemTime();

IF f_Trig_HB.Q THEN
	IF intCount>50 OR intCount<0 THEN
		intCount:=0;
	END_IF
	stringArray_Last_HB[intCount] := prg_SystemTime.stringSystemTime_ms;
	intCount := intCount+1;
END_IF

time_Temp := fbCom.fbTimerHB.ET;

// fbMqttClient.bError OR fbJsonRead.bError OR fbGetTime.ERR
count_u(
	CU:= fbCom.fbJsonRead.bErrorIntern, 
	RESET:= , 
	PV:= , 
	Q=> , 
	CV=> ); 
count_u1(
	CU:= fbCom.fbJsonRead.bError, 
	RESET:= , 
	PV:= , 
	Q=> , 
	CV=> );
count_u2(
	CU:= fbCom.fbJsonRead.bDetected, 
	RESET:= , 
	PV:= , 
	Q=> , 
	CV=> );  
IF 	fbCom.fbJsonRead.bError THEN
	eErrorMessage_Read := fbCom.fbJsonRead.eErrorMessage_Out;
END_IF

arrErrorIntern := fbCom.fbJsonRead.arrErrorIntern;

END_PROGRAM

// ---- POUs/prgRWEffIO.TcPOU
PROGRAM prgRWEffIO
VAR
	fbRW1		: FB_ReadWrite_V2;
END_VAR

fbRW1(	eUploadType := eSelectDataUploadType.e_Change_Intervall1min,
		bBusy=> , 
		bError=> , 
		udiErrorCodeOut=> , 
		eErrorReadWrite_Out=> );

END_PROGRAM
